{attribute 'GeneratedUsingTerminal: EK1122-0000-0018'}
{attribute addProperty BoxType "EK1122-0000-0018"}
{attribute addProperty Id "Beckhoff_ER4xxxsub_EK1100EK1100_1FC0878B2A_0001_ER4174_0002_0016ER4174_D2A7C9B719A_0002_ER4174_0002_0019ER4174_D2A7C9B719A_0003_ER4374_0002_0018ER4374_6231FEFD36A_0004_ER4374_0002_0019ER4374_6231FEFD36"}
{attribute addProperty CRC "3086166838"}
{attribute addProperty Size "112"}
TYPE Beckhoff_ER4xxxEK1122_B7F32B36 EXTENDS EK1122_1FC0878B :
STRUCT
	{attribute addProperty Name "Beckhoff_ER4xxxsub_EK1100"}
	{attribute addProperty PreviousPort "Beckhoff ER4xxxEK1122 : D"}
	Beckhoff_ER4xxxsub_EK1100 : EK1100_1FC0878B;
	{attribute addProperty Name "A_0001_ER4174_0002_0016"}
	{attribute addProperty PreviousPort "Beckhoff ER4xxxsub EK1100 : C"}
	A_0001_ER4174_0002_0016 : ER4174_D2A7C9B7;
	{attribute addProperty Name "A_0002_ER4174_0002_0019"}
	{attribute addProperty PreviousPort "A_0001(ER4174-0002-0016) : B"}
	A_0002_ER4174_0002_0019 : ER4174_D2A7C9B7;
	{attribute addProperty Name "A_0003_ER4374_0002_0018"}
	{attribute addProperty PreviousPort "A_0002(ER4174-0002-0019) : B"}
	A_0003_ER4374_0002_0018 : ER4374_6231FEFD;
	{attribute addProperty Name "A_0004_ER4374_0002_0019"}
	{attribute addProperty PreviousPort "A_0003(ER4374-0002-0018) : B"}
	A_0004_ER4374_0002_0019 : ER4374_6231FEFD;
END_STRUCT
END_TYPE

(* stored: Version 1.2.0.0, ProductVersion 3.1.4024.9
   DUT Beckhoff_ER4xxxEK1122_B7F32B36: Id {93e85a68-e23a-4a02-b8d5-fd152b068175} *)
